// TIA Portal V17 export
// export: Created 2024-09-02T12:49:55.8162824Z, ExportSetting WithDefaults, DisplayName Totally Integrated Automation Portal, DisplayVersion V17, DisplayName TIA Portal Openness, DisplayVersion V17, DisplayName TIA Portal Version Control Interface, DisplayVersion V17, DisplayName STEP 7 Professional, DisplayVersion V17, DisplayName STEP 7 Safety, DisplayVersion V17, DisplayName WinCC Professional, DisplayVersion V17
FUNCTION "SysFC_HMI_HandMovements" : Void   // FC250, LAD
TITLE = Supply hand line / Versorgung Handzeile
{ S7_Optimized_Access := 'TRUE' }
AUTHOR : OlegFuehrus
FAMILY : HMI
NAME : HMI
VERSION : 0.1
// stored: AutoNumber true, IsIECCheckEnabled false, SetENOAutomatically false, UDAEnableTagReadback false
   VAR_INPUT
      Line : Int;   // Zeile (1..348) / Line (1. . 348)
      Control_WORK : Bool;   // Ansteuerung Arbeiststellung / Control of working position
      Control_HOME : Bool;   // Ansteuerung Grundstellung / Control Basic position
      Position_WORK : Bool;   // Endlage Arbeitsstellung / End position Working position
      Position_HOME : Bool;   // Endlage Arbeitsstellung / End position Working position
      Position : LReal;   // Positionsanzeige / position display
      "Hide Pos." : Bool;   // Position ausblenden / Hide position
      "Hide Left Arrow" : Bool;   // Pfeil Links ausblenden / Hide left arrow
      "Hide Right Arrow" : Bool;   // Pfeil Rechts ausblenden / Hide left arrow
      ACK : Bool;   // Quitt
      "ParityFault Time" : Time;   // Überschneidungszeit Paarfehler (0..2s) / Overlap time pair error (0. . 2s)
   END_VAR
   VAR_OUTPUT
      ParityFault : Bool;   // Paarfehler / pair error
      ConfigFault : Bool;   // Configurationsfehler / configuration error
   END_VAR
   VAR_IN_OUT
      LTLL_Config : "LTLL_typeConfig";
      LTLL_Data : "LTLL_typeData";
      LTLL_S7GConfig : "LTLL_typeManualGraphConfig";
      SYS_LineHand : "TypeStepsHand";
   END_VAR
   VAR_TEMP
      t_RetVal : Word;
      t_VKE0 : Bool;
      t_VKE1 : Bool;
      t_ConfigFault : Bool;
      t_ConfigFaultNr : Int;
      t_Line : Int;
      t_Line_UInt : UInt;
      t_Btn_Left : Bool;
      t_Btn_Right : Bool;
      t_secure_bit_ok : Bool;
      t_ErrID : Word;
      t_loop : Int;
      t_Pointer : Int;
   END_VAR
   VAR_TEMP   // added for the SCL form of the ladder/FBD networks
      _w1 : Bool;
   END_VAR
BEGIN

REGION Network 1: VKE0
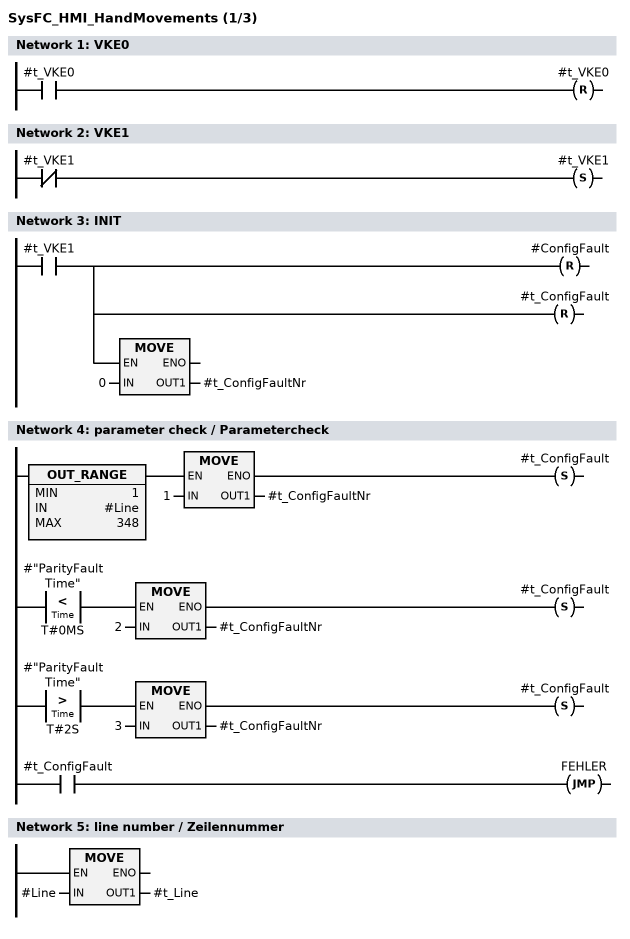
   RUNG wire#powerrail
      Contact( #t_VKE0 )
      R_Coil( #t_VKE0 )
   END_RUNG
   // the same network as SCL:
   IF #t_VKE0 THEN #t_VKE0 := FALSE; END_IF;
END_REGION

REGION Network 2: VKE1
   RUNG wire#powerrail
      I_Contact( #t_VKE1 )
      S_Coil( #t_VKE1 )
   END_RUNG
   // the same network as SCL:
   IF NOT #t_VKE1 THEN #t_VKE1 := TRUE; END_IF;
END_REGION

REGION Network 3: INIT
   RUNG wire#powerrail
      Contact( #t_VKE1 )
      wire#w1
      R_Coil( #ConfigFault )
   END_RUNG
   RUNG wire#w1
      R_Coil( #t_ConfigFault )
   END_RUNG
   RUNG wire#w1
      Move(in := 0, out1 => #t_ConfigFaultNr)
   END_RUNG
   // the same network as SCL:
   IF #t_VKE1 THEN
       #ConfigFault := FALSE;
       #t_ConfigFault := FALSE;
       #t_ConfigFaultNr := 0;
   END_IF;
END_REGION

REGION Network 4: parameter check / Parametercheck
   IF (#Line < 1) OR (#Line > 348) THEN
       #t_ConfigFaultNr := 1;
       #t_ConfigFault := TRUE;
   END_IF;
   IF #"ParityFault Time" < T#0MS THEN
       #t_ConfigFaultNr := 2;
       #t_ConfigFault := TRUE;
   END_IF;
   IF #"ParityFault Time" > T#2S THEN
       #t_ConfigFaultNr := 3;
       #t_ConfigFault := TRUE;
   END_IF;
   IF #t_ConfigFault THEN GOTO FEHLER; END_IF;
END_REGION

REGION Network 5: line number / Zeilennummer
   RUNG wire#powerrail
      Move(in := #Line, out1 => #t_Line)
   END_RUNG
   // the same network as SCL:
   #t_Line := #Line;
END_REGION

REGION Network 6: Supply line / Zeile versorgen
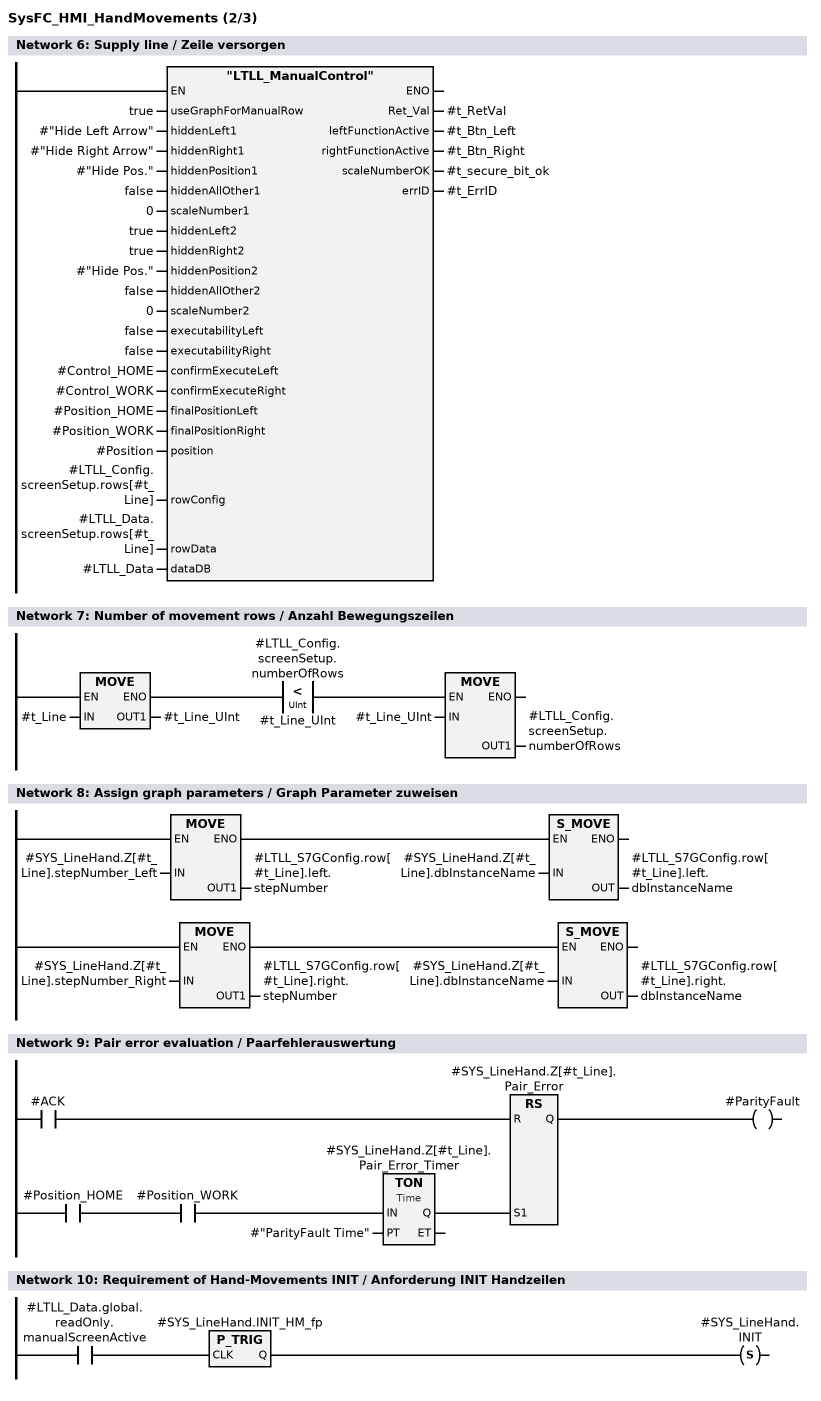
   RUNG wire#powerrail
      "LTLL_ManualControl"(useGraphForManualRow := true, hiddenLeft1 := #"Hide Left Arrow", hiddenRight1 := #"Hide Right Arrow", hiddenPosition1 := #"Hide Pos.", hiddenAllOther1 := false, scaleNumber1 := 0, hiddenLeft2 := true, hiddenRight2 := true, hiddenPosition2 := #"Hide Pos.", hiddenAllOther2 := false, scaleNumber2 := 0, executabilityLeft := false, executabilityRight := false, confirmExecuteLeft := #Control_HOME, confirmExecuteRight := #Control_WORK, finalPositionLeft := #Position_HOME, finalPositionRight := #Position_WORK, position := #Position, rowConfig := #LTLL_Config.screenSetup.rows[#t_Line], rowData := #LTLL_Data.screenSetup.rows[#t_Line], dataDB := #LTLL_Data, Ret_Val => #t_RetVal, leftFunctionActive => #t_Btn_Left, rightFunctionActive => #t_Btn_Right, scaleNumberOK => #t_secure_bit_ok, errID => #t_ErrID)
   END_RUNG
   // the same network as SCL:
   #t_RetVal := "LTLL_ManualControl"(useGraphForManualRow := true,
                           hiddenLeft1 := #"Hide Left Arrow",
                           hiddenRight1 := #"Hide Right Arrow",
                           hiddenPosition1 := #"Hide Pos.",
                           hiddenAllOther1 := false,
                           scaleNumber1 := 0,
                           hiddenLeft2 := true,
                           hiddenRight2 := true,
                           hiddenPosition2 := #"Hide Pos.",
                           hiddenAllOther2 := false,
                           scaleNumber2 := 0,
                           executabilityLeft := false,
                           executabilityRight := false,
                           confirmExecuteLeft := #Control_HOME,
                           confirmExecuteRight := #Control_WORK,
                           finalPositionLeft := #Position_HOME,
                           finalPositionRight := #Position_WORK,
                           position := #Position,
                           rowConfig := #LTLL_Config.screenSetup.rows[#t_Line],
                           rowData := #LTLL_Data.screenSetup.rows[#t_Line],
                           dataDB := #LTLL_Data,
                           leftFunctionActive => #t_Btn_Left,
                           rightFunctionActive => #t_Btn_Right,
                           scaleNumberOK => #t_secure_bit_ok,
                           errID => #t_ErrID);
END_REGION

REGION Network 7: Number of movement rows / Anzahl Bewegungszeilen
   RUNG wire#powerrail
      Move(in := #t_Line, out1 => #t_Line_UInt)
      { S7_Templates := "SrcType := UInt" } LT_Contact(in1 := #LTLL_Config.screenSetup.numberOfRows, in2 := #t_Line_UInt)
      Move(in := #t_Line_UInt, out1 => #LTLL_Config.screenSetup.numberOfRows)
   END_RUNG
   // the same network as SCL:
   #t_Line_UInt := #t_Line;
   IF #LTLL_Config.screenSetup.numberOfRows < #t_Line_UInt THEN
       #LTLL_Config.screenSetup.numberOfRows := #t_Line_UInt;
   END_IF;
END_REGION

REGION Network 8: Assign graph parameters / Graph Parameter zuweisen
   RUNG wire#powerrail
      Move(in := #SYS_LineHand.Z[#t_Line].stepNumber_Left, out1 => #LTLL_S7GConfig.row[#t_Line].left.stepNumber)
      S_Move(in := #SYS_LineHand.Z[#t_Line].dbInstanceName, out => #LTLL_S7GConfig.row[#t_Line].left.dbInstanceName)
   END_RUNG
   RUNG wire#powerrail
      Move(in := #SYS_LineHand.Z[#t_Line].stepNumber_Right, out1 => #LTLL_S7GConfig.row[#t_Line].right.stepNumber)
      S_Move(in := #SYS_LineHand.Z[#t_Line].dbInstanceName, out => #LTLL_S7GConfig.row[#t_Line].right.dbInstanceName)
   END_RUNG
   // the same network as SCL:
   #LTLL_S7GConfig.row[#t_Line].left.stepNumber := #SYS_LineHand.Z[#t_Line].stepNumber_Left;
   #LTLL_S7GConfig.row[#t_Line].left.dbInstanceName := #SYS_LineHand.Z[#t_Line].dbInstanceName;
   #LTLL_S7GConfig.row[#t_Line].right.stepNumber := #SYS_LineHand.Z[#t_Line].stepNumber_Right;
   #LTLL_S7GConfig.row[#t_Line].right.dbInstanceName := #SYS_LineHand.Z[#t_Line].dbInstanceName;
END_REGION

REGION Network 9: Pair error evaluation / Paarfehlerauswertung
   RUNG wire#powerrail
      Contact( #ACK )
      S_RS(operand := #SYS_LineHand.Z[#t_Line].Pair_Error, s1 := wire#w1)
      Coil( #ParityFault )
   END_RUNG
   RUNG wire#powerrail
      Contact( #Position_HOME )
      Contact( #Position_WORK )
      { S7_Templates := "time_type := Time" } #SYS_LineHand.Z[#t_Line].Pair_Error_Timer.TON(pt := #"ParityFault Time", et =>)
   END_RUNG wire#w1
   // the same network as SCL:
   #SYS_LineHand.Z[#t_Line].Pair_Error_Timer.TON(IN := #Position_HOME AND #Position_WORK,
                           PT := #"ParityFault Time");
   #_w1 := #SYS_LineHand.Z[#t_Line].Pair_Error_Timer.Q;
   IF #ACK THEN
       #SYS_LineHand.Z[#t_Line].Pair_Error := FALSE;   // RS flip-flop
   END_IF;
   IF #_w1 THEN #SYS_LineHand.Z[#t_Line].Pair_Error := TRUE; END_IF;
   #ParityFault := #SYS_LineHand.Z[#t_Line].Pair_Error;
END_REGION

REGION Network 10: Requirement of Hand-Movements INIT / Anforderung INIT Handzeilen
   RUNG wire#powerrail
      Contact( #LTLL_Data.global.readOnly.manualScreenActive )
      P_Trig( #SYS_LineHand.INIT_HM_fp )
      S_Coil( #SYS_LineHand.INIT )
   END_RUNG
   // the same network as SCL:
   #_w1 := #LTLL_Data.global.readOnly.manualScreenActive AND NOT #SYS_LineHand.INIT_HM_fp;   // rising edge
   #SYS_LineHand.INIT_HM_fp := #LTLL_Data.global.readOnly.manualScreenActive;
   IF #_w1 THEN #SYS_LineHand.INIT := TRUE; END_IF;
END_REGION

REGION Network 11 (SCL): INIT hand lines / INIT Handzeilen
   IF  #SYS_LineHand.INIT THEN
       FOR #t_Pointer := 1 TO 348 BY 1 DO
           #LTLL_Config.screenSetup.rows[#t_Pointer].configs[0].hiddenLeft := true;
           #LTLL_Config.screenSetup.rows[#t_Pointer].configs[0].hiddenRight := true;
           #LTLL_Config.screenSetup.rows[#t_Pointer].configs[0].hiddenPosition := true;
           #LTLL_Config.screenSetup.rows[#t_Pointer].configs[0].hiddenAllOther := true;
           #LTLL_Config.screenSetup.rows[#t_Pointer].configs[1].hiddenLeft := true;
           #LTLL_Config.screenSetup.rows[#t_Pointer].configs[1].hiddenRight := true;
           #LTLL_Config.screenSetup.rows[#t_Pointer].configs[1].hiddenPosition := true;
           #LTLL_Config.screenSetup.rows[#t_Pointer].configs[1].hiddenAllOther := true;

           #LTLL_Data.screenSetup.rows[#t_Pointer].runtimeInterface.executabilityLeft := false;
           #LTLL_Data.screenSetup.rows[#t_Pointer].runtimeInterface.executabilityRight := false;
           #LTLL_Data.screenSetup.rows[#t_Pointer].runtimeInterface.confirmExecuteLeft := false;
           #LTLL_Data.screenSetup.rows[#t_Pointer].runtimeInterface.confirmExecuteRight := false;
           #LTLL_Data.screenSetup.rows[#t_Pointer].runtimeInterface.finalPositionLeft := false;
           #LTLL_Data.screenSetup.rows[#t_Pointer].runtimeInterface.finalPositionRight := false;
       END_FOR;
       #SYS_LineHand.INIT := false;
   END_IF;
END_REGION

REGION Network 12: Error evaluation / Fehlerauswertung
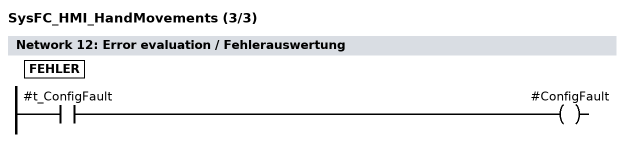
   Label( FEHLER )
   RUNG wire#powerrail
      Contact( #t_ConfigFault )
      Coil( #ConfigFault )
   END_RUNG
   // the same network as SCL:
   FEHLER:
   #ConfigFault := #t_ConfigFault;
END_REGION
END_FUNCTION
